// TwinCAT 3 PLC project Sample03
// ProgramVersion: 3.1.0.8
// libraries:
//   Tc2_Standard, * (Beckhoff Automation GmbH)
//   Tc2_System, * (Beckhoff Automation GmbH)
//   Tc2_Utilities, * (Beckhoff Automation GmbH)
//   Tc3_Interfaces, * (Beckhoff Automation GmbH)
//   Tc3_MemMan, * (Beckhoff Automation GmbH)
//   Tc3_Module, * (Beckhoff Automation GmbH)
// project tree:
//   / PlcTask.TcTTO
//   POUs/ FB_DatabaseLoggerFactory.TcPOU, MAIN.TcPOU, FB_SQLServerLogger.TcPOU
//   POUs/PLC-Library/ FB_AbstractLoggerFactory.TcPOU, FB_CsvLogger.TcPOU, FB_FileLoggerFactory.TcPOU, FB_Logger.TcPOU, FB_TxtLogger.TcPOU, FB_XmlLogger.TcPOU, ILogger.TcIO
// real-time tasks:
//   TASK PlcTask: cycle T#10ms, priority 20, ADS port 350

CONFIGURATION Sample03
    RESOURCE PLC ON TwinCAT3
        TASK PlcTask(INTERVAL := T#10ms, PRIORITY := 20);
        PROGRAM MAIN WITH PlcTask : MAIN;
    END_RESOURCE
END_CONFIGURATION

// ---- POUs/PLC-Library/ILogger.TcIO
INTERFACE ILogger

METHOD Write : STRING
VAR_INPUT
	sMsg	: STRING;
END_VAR
END_METHOD

END_INTERFACE

// ---- POUs/MAIN.TcPOU
PROGRAM MAIN
VAR
    fbDatabaseLoggerFactory  : FB_DatabaseLoggerFactory('MyDatabase', 'User', 'Password');
    refDatabaseLoggerFactory : REFERENCE TO FB_DatabaseLoggerFactory := fbDatabaseLoggerFactory;
    fbLogger                 : FB_Logger(refDatabaseLoggerFactory);	
    sRetMsg                  : STRING;
END_VAR

sRetMsg := fbLogger.Write('Hello');

END_PROGRAM

// ---- POUs/FB_DatabaseLoggerFactory.TcPOU
FUNCTION_BLOCK INTERNAL FB_DatabaseLoggerFactory EXTENDS FB_AbstractLoggerFactory
VAR
	pSQLServerLogger  : POINTER TO FB_SQLServerLogger;
    ipLogger          : ILogger := 0;
END_VAR

METHOD FB_exit : BOOL
VAR_INPUT
	bInCopyCode : BOOL; // if TRUE, the exit method is called for exiting an instance that is copied afterwards (online change).
END_VAR
IF (pSQLServerLogger <> 0) THEN
	__DELETE(pSQLServerLogger);
	pSQLServerLogger := 0;
END_IF
END_METHOD

METHOD FB_init : BOOL
VAR_INPUT
	bInitRetains : BOOL; // if TRUE, the retain variables are initialized (warm start / cold start)
	bInCopyCode  : BOOL;  // if TRUE, the instance afterwards gets moved into the copy code (online change)
	sDataSource  : STRING;
	sPassword    : STRING;
	sUser        : STRING;
END_VAR
pSQLServerLogger := __NEW(FB_SQLServerLogger);
ipLogger := pSQLServerLogger^;
END_METHOD

METHOD PUBLIC GetLogger : ILogger
VAR_INPUT
END_VAR
GetLogger := ipLogger;
END_METHOD

END_FUNCTION_BLOCK

// ---- POUs/PLC-Library/FB_AbstractLoggerFactory.TcPOU
FUNCTION_BLOCK public FB_AbstractLoggerFactory
VAR_INPUT
END_VAR
VAR_OUTPUT
END_VAR
VAR
END_VAR

METHOD PUBLIC GetLogger : ILogger
VAR_INPUT
END_VAR
;
END_METHOD

END_FUNCTION_BLOCK

// ---- POUs/FB_SQLServerLogger.TcPOU
{attribute 'enable_dynamic_creation'}
FUNCTION_BLOCK INTERNAL FB_SQLServerLogger IMPLEMENTS ILogger
VAR_INPUT
END_VAR
VAR_OUTPUT
END_VAR
VAR
END_VAR

METHOD PUBLIC Write : STRING
VAR_INPUT
	sMsg	: string;
END_VAR
Write := CONCAT('DatabaseLogger: ', sMsg);
END_METHOD

END_FUNCTION_BLOCK

// ---- POUs/PLC-Library/FB_Logger.TcPOU
FUNCTION_BLOCK PUBLIC FB_Logger
VAR
	ipLogger : ILogger;
END_VAR

METHOD FB_init : BOOL
VAR_INPUT
	bInitRetains       : BOOL; // if TRUE, the retain variables are initialized (warm start / cold start)
	bInCopyCode        : BOOL;  // if TRUE, the instance afterwards gets moved into the copy code (online change)
	refLoggerFactory   : REFERENCE TO FB_AbstractLoggerFactory;
END_VAR
IF (__ISVALIDREF(refLoggerFactory)) THEN
	ipLogger := refLoggerFactory.GetLogger();
ELSE
	ipLogger := 0;
END_IF
END_METHOD

METHOD PUBLIC Write : STRING
VAR_INPUT
	message 		 : STRING;
END_VAR
Write := 'Error';
IF (ipLogger <> 0) THEN
	Write := ipLogger.Write(message);
END_IF
END_METHOD

END_FUNCTION_BLOCK

// ---- POUs/PLC-Library/FB_CsvLogger.TcPOU
{attribute 'enable_dynamic_creation'}
FUNCTION_BLOCK INTERNAL FB_CsvLogger IMPLEMENTS ILogger
VAR_INPUT
END_VAR
VAR_OUTPUT
END_VAR
VAR
END_VAR

METHOD PUBLIC Write : STRING
VAR_INPUT
	sMsg : string;
END_VAR
Write := CONCAT('CsvLogger: ', sMsg);
END_METHOD

END_FUNCTION_BLOCK

// ---- POUs/PLC-Library/FB_FileLoggerFactory.TcPOU
FUNCTION_BLOCK INTERNAL FB_FileLoggerFactory EXTENDS FB_AbstractLoggerFactory
VAR
	pTxtLogger  : POINTER TO FB_TxtLogger;
	pCsvLogger  : POINTER TO FB_CsvLogger;
	pXmlLogger  : POINTER TO FB_XmlLogger;
    ipLogger    : ILogger := 0;
END_VAR

METHOD FB_init : BOOL
VAR_INPUT
	bInitRetains : BOOL; // if TRUE, the retain variables are initialized (warm start / cold start)
	bInCopyCode  : BOOL;  // if TRUE, the instance afterwards gets moved into the copy code (online change)
	sFilename    : STRING;
END_VAR
VAR
	sFilenameExtension : STRING;
END_VAR
sFilenameExtension := F_ToLCase(RIGHT(sFilename, 3));
IF (sFilenameExtension = 'txt') THEN
    pTxtLogger := __NEW(FB_TxtLogger);
    ipLogger := pTxtLogger^;
ELSIF (sFilenameExtension = 'csv') THEN
    pCsvLogger := __NEW(FB_CsvLogger);
    ipLogger := pCsvLogger^;
ELSIF (sFilenameExtension = 'xml') THEN
    pXmlLogger := __NEW(FB_XmlLogger);
    ipLogger := pXmlLogger^;
ELSE
    ipLogger := 0;
END_IF
END_METHOD

METHOD FB_exit : BOOL
VAR_INPUT
	bInCopyCode : BOOL; // if TRUE, the exit method is called for exiting an instance that is copied afterwards (online change).
END_VAR
IF (pTxtLogger <> 0) THEN
	__DELETE(pTxtLogger);
	pTxtLogger := 0;
END_IF

IF (pCsvLogger <> 0) THEN
	__DELETE(pCsvLogger);
	pCsvLogger := 0;
END_IF

IF (pXmlLogger <> 0) THEN
	__DELETE(pXmlLogger);
	pXmlLogger := 0;
END_IF
END_METHOD

METHOD PUBLIC GetLogger : ILogger
VAR_INPUT
END_VAR
GetLogger := ipLogger;
END_METHOD

END_FUNCTION_BLOCK

// ---- POUs/PLC-Library/FB_TxtLogger.TcPOU
{attribute 'enable_dynamic_creation'}
FUNCTION_BLOCK INTERNAL FB_TxtLogger IMPLEMENTS ILogger
VAR_INPUT
END_VAR
VAR_OUTPUT
END_VAR
VAR
END_VAR

METHOD PUBLIC Write : STRING
VAR_INPUT
	sMsg : STRING;
END_VAR
Write := CONCAT('TxtLogger: ', sMsg);
END_METHOD

END_FUNCTION_BLOCK

// ---- POUs/PLC-Library/FB_XmlLogger.TcPOU
{attribute 'enable_dynamic_creation'}
FUNCTION_BLOCK INTERNAL FB_XmlLogger IMPLEMENTS ILogger
VAR_INPUT
END_VAR
VAR_OUTPUT
END_VAR
VAR
END_VAR

METHOD PUBLIC Write : STRING
VAR_INPUT
	sMsg	: string;
END_VAR
Write := CONCAT('XmlLogger: ', sMsg);
END_METHOD

END_FUNCTION_BLOCK
